(* CODESYS project StateTrafficLight.project

Project tree, tasks and I/O mapping:
  Device : CODESYS Control Win V3, 3S - Smart Software Solutions GmbH, order no. 305021, version 3.5.10.40
    application Application
      libraries: Standard, * (System)
      task MainTask (cyclic, interval t#20ms, priority 1) calls PLC_PRG
      task VISU_TASK (cyclic, interval 100 ms, priority 31) calls VisuElems.Visu_Prg
      program PLC_PRG [FBD]
      function block TrafficLight [SFC]: Green_state_entry, Yellow_State_entry, Red_State_entry, Green_state_exit, Yellow_State_exit, Red_State_exit, Init_active
      visualisation Visualization
      function block BlinkingYellow_Sequencial [SFC]: Init_active, Blink_entry
  text list GlobalTextList
*)

// Device/Application/PLC_PRG
PROGRAM PLC_PRG
VAR
	TrafficLight_0: TrafficLight;
	Contact1: BOOL := FALSE;
	yellow_led: BOOL := FALSE;
	green_led: BOOL := FALSE;
	red_led: BOOL := FALSE;
	flag: BOOL := FALSE;
	BlinkingYellow_Sequencial_0: BlinkingYellow_Sequencial;
	yellow_led2: BOOL := FALSE;
END_VAR

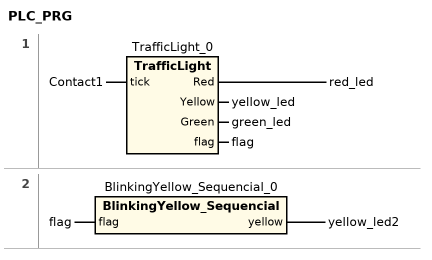
// NETWORK 1
TrafficLight_0(tick := Contact1, Yellow => yellow_led, Green => green_led, flag => flag); // TrafficLight
red_led := TrafficLight_0.Red;

// NETWORK 2
BlinkingYellow_Sequencial_0(flag := flag); // BlinkingYellow_Sequencial
yellow_led2 := BlinkingYellow_Sequencial_0.yellow;

END_PROGRAM

// Device/Application/TrafficLight
FUNCTION_BLOCK TrafficLight
VAR_INPUT
	tick : BOOL := FALSE;
END_VAR

VAR_OUTPUT
	Red : BOOL := FALSE;
	Yellow : BOOL := FALSE;
	Green : BOOL := FALSE;
	flag :BOOL := FALSE;
	noflag :BOOL := TRUE;
END_VAR

VAR
	i : INT := 0;
END_VAR

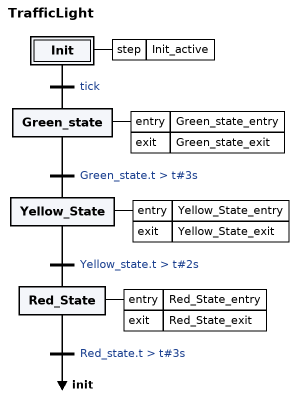
INITIAL_STEP Init:
    Init_active(N);  // step action
END_STEP
TRANSITION FROM Init TO Green_state
    := tick;
END_TRANSITION
STEP Green_state:
    Green_state_entry(P1);  // entry action
    Green_state_exit(P0);  // exit action
END_STEP
TRANSITION FROM Green_state TO Yellow_State
    := Green_state.t > t#3s;
END_TRANSITION
STEP Yellow_State:
    Yellow_State_entry(P1);  // entry action
    Yellow_State_exit(P0);  // exit action
END_STEP
TRANSITION FROM Yellow_State TO Red_State
    := Yellow_state.t > t#2s;
END_TRANSITION
STEP Red_State:
    Red_State_entry(P1);  // entry action
    Red_State_exit(P0);  // exit action
END_STEP
TRANSITION FROM Red_State TO init
    := Red_state.t > t#3s;
END_TRANSITION

ACTION Green_state_entry:
IF NOT FLAG AND tick THEN
	green := TRUE;
	i:=i+1;
END_IF
END_ACTION

ACTION Yellow_State_entry:
IF NOT FLAG AND tick THEN
	yellow := TRUE;
END_IF
END_ACTION

ACTION Red_State_entry:
IF NOT FLAG AND tick THEN
	red := TRUE;
END_IF
END_ACTION

ACTION Green_state_exit:
green := FALSE;
IF NOT tick THEN
	flag := FALSE;
END_IF
IF i > 4 AND tick THEN;
	flag := TRUE;
END_IF
END_ACTION

ACTION Yellow_State_exit:
yellow := FALSE;
END_ACTION

ACTION Red_State_exit:
red:=FALSE;
END_ACTION

ACTION Init_active:
IF NOT tick THEN
	flag := FALSE;
	i := 0;
	red := FALSE;
	yellow := FALSE;
	green := FALSE;
END_IF
END_ACTION

END_FUNCTION_BLOCK

// Device/Application/BlinkingYellow_Sequencial
FUNCTION_BLOCK BlinkingYellow_Sequencial
VAR_INPUT
	flag : BOOL := FALSE;
END_VAR

VAR_OUTPUT
	yellow : BOOL ;
END_VAR
VAR
END_VAR

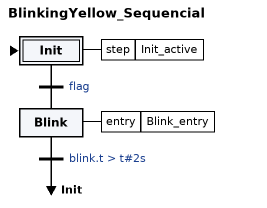
INITIAL_STEP Init:
    Init_active(N);  // step action
END_STEP
TRANSITION FROM Init TO Blink
    := flag;
END_TRANSITION
STEP Blink:
    Blink_entry(P1);  // entry action
END_STEP
TRANSITION FROM Blink TO Init
    := blink.t > t#2s;
END_TRANSITION

ACTION Init_active:
IF NOT flag THEN 
	yellow := FALSE;
END_IF
END_ACTION

ACTION Blink_entry:
IF flag THEN
	yellow := NOT yellow;
END_IF
END_ACTION

END_FUNCTION_BLOCK

// Device/Application/Visualization
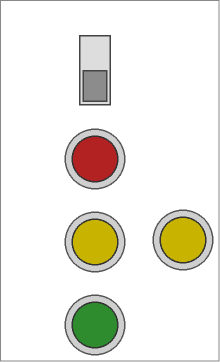
VISUALIZATION Visualization  // 220x362
    Lamp1 (60,124 70x70), variable: PLC_PRG.red_led, style: Lamp-Lamp1-Red
    Lamp1 (60,207 70x70), variable: PLC_PRG.yellow_led, style: Lamp-Lamp1-Yellow
    Lamp1 (60,290 70x70), variable: PLC_PRG.green_led, style: Lamp-Lamp1-Green
    DipSwitch (60,35 70x70), variable: PLC_PRG.Contact1, behaviour: TOGGLE, style: Switch-DipSwitch-Gray
    Lamp1 (148,205 70x70), variable: PLC_PRG.yellow_led2, style: Lamp-Lamp1-Yellow
END_VISUALIZATION
